FUNCTION_BLOCK FB_FalliblePublic_Test EXTENDS FB_TestSuiteExtended


TestSetErrorGetErrorExpectErrorStatus();


METHOD PRIVATE TestSetErrorGetErrorExpectErrorStatus
VAR
    sMsg : T_MaxString;
    fbFalliblePublic : FB_FalliblePublic;
END_VAR

TEST('TestSetErrorGetErrorExpectErrorStatus');

// Test fixture
sMsg := 'Error';
fbFalliblePublic.SetError(Msg := sMsg);

// Subject Under Test
AssertTrue(
    Condition := fbFalliblePublic.GetError(),
    Message := 'Expected GetError to be true, but it was false.'
);

AssertTrue(
    Condition := fbFalliblePublic.GetErrorMsg() = sMsg,
    Message := 'Expected error message to match what it was set to.'
);

TEST_FINISHED();
END_METHOD

END_FUNCTION_BLOCK

(* stored: Version 1.1.0.1
   POU FB_FalliblePublic_Test: Id {1c35488e-a1b4-4740-8d28-946a9629b058}, SpecialFunc None
   Method TestSetErrorGetErrorExpectErrorStatus: Id {2a272c6d-58f1-41c7-953d-9cf107ecb189} *)
